PROGRAM init_axes
VAR
	states : ARRAY[0..3] OF INT := 0;
	errors : ARRAY[0..3] OF BOOL := FALSE;
	
	mcPowers : ARRAY[0..3] OF MC_Power;
	mcSetPositions : ARRAY[0..3] OF MC_SetPosition;
	mcMoveAbsolutes : ARRAY[0..3] OF MC_MoveAbsolute;
	i: INT;
END_VAR


FOR i := 0 TO 3 DO
	main.axes[i].ReadStatus();
	CASE states[i] OF
		0:
			// activate motors
			mcPowers[i](
				Axis := main.axes[i],
				Enable := TRUE,
				Enable_Positive := TRUE,
				Enable_Negative := TRUE,
				BufferMode := MC_Aborting
			);
			states[i] := 1;
		1:
			// check for error
			IF mcPowers[i].Active THEN
				states[i] := 2;
			ELSE
				states[i] := 100;
			END_IF
		2:
			// constantly set current position to 0
			mcSetPositions[i](
				Axis:= main.axes[i], 
				Execute:= TRUE, 
				Position:= 0.0
			);
		100:
			errors[i] := TRUE;
	END_CASE
END_FOR

END_PROGRAM

(* stored: Version 1.1.0.1, ProductVersion 3.1.4024.12
   POU init_axes: Id {0153cdfc-a178-4b6b-918c-07d5d7034082}, SpecialFunc None *)
